// Mitsubishi GX Works2 project: shrimp_load_v02   PLC: FX3G
// Carga de PLC para monitoreo de piscina de camarones

PROGRAM MAIN
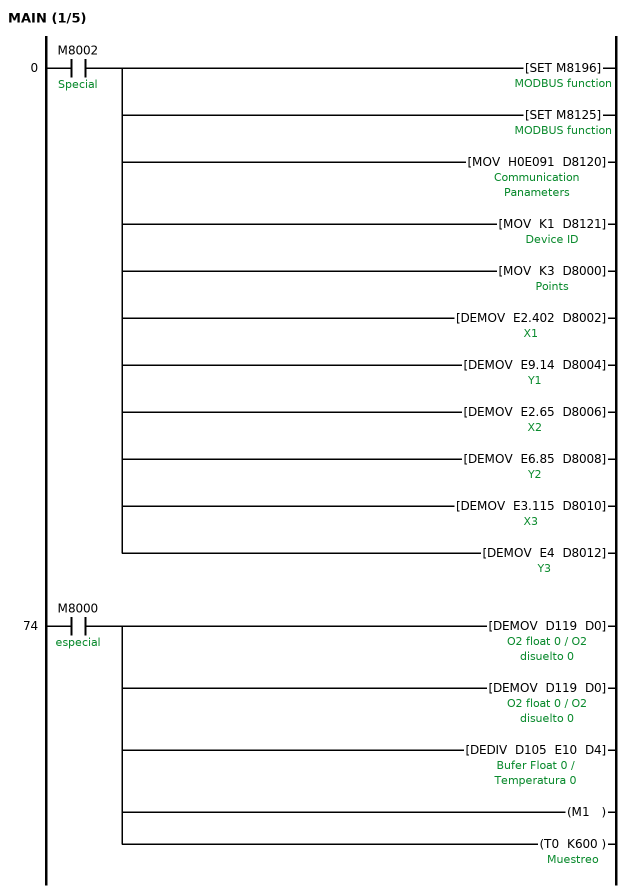
0     LD      M8002  ; Special
      SET     M8196  ; MODBUS function
      SET     M8125  ; MODBUS function
      MOV     H0E091 D8120  ; Communication Panameters
      MOV     K1 D8121  ; Device ID
      MOV     K3 D8000  ; Points
      DEMOV   E2.402 D8002  ; X1
      DEMOV   E9.14 D8004  ; Y1
      DEMOV   E2.65 D8006  ; X2
      DEMOV   E6.85 D8008  ; Y2
      DEMOV   E3.115 D8010  ; X3
      DEMOV   E4 D8012  ; Y3
74    LD      M8000  ; especial
      DEMOV   D119 D0  ; O2 float 0 / O2 disuelto 0
      DEMOV   D119 D0
      DEDIV   D105 E10 D4  ; Bufer Float 0 / Temperatura 0
      OUT     M1
      OUT     T0 K600  ; Muestreo
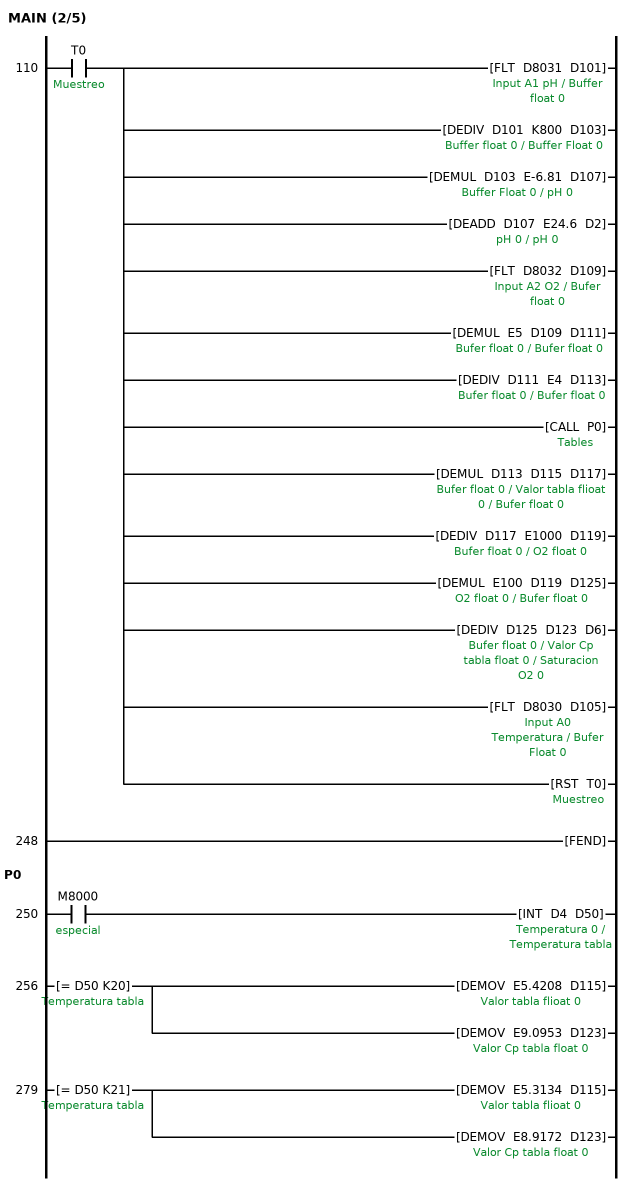
110   LD      T0  ; Muestreo
      FLT     D8031 D101  ; Input A1 pH / Buffer float 0
      DEDIV   D101 K800 D103  ; Buffer Float 0
      DEMUL   D103 E-6.81 D107  ; pH 0
      DEADD   D107 E24.6 D2  ; pH 0
      FLT     D8032 D109  ; Input A2 O2 / Bufer float 0
      DEMUL   E5 D109 D111  ; Bufer float 0
      DEDIV   D111 E4 D113  ; Bufer float 0
      CALL    P0  ; Tables
      DEMUL   D113 D115 D117  ; Valor tabla flioat 0 / Bufer float 0
      DEDIV   D117 E1000 D119
      DEMUL   E100 D119 D125  ; Bufer float 0
      DEDIV   D125 D123 D6  ; Valor Cp tabla float 0 / Saturacion O2 0
      FLT     D8030 D105  ; Input A0 Temperatura
      RST     T0  ; Muestreo
248   FEND
      P0
250   LD      M8000  ; especial
      INT     D4 D50  ; Temperatura tabla
256   LD=     D50 K20  ; Temperatura tabla
      DEMOV   E5.4208 D115
      DEMOV   E9.0953 D123
279   LD=     D50 K21  ; Temperatura tabla
      DEMOV   E5.3134 D115
      DEMOV   E8.9172 D123
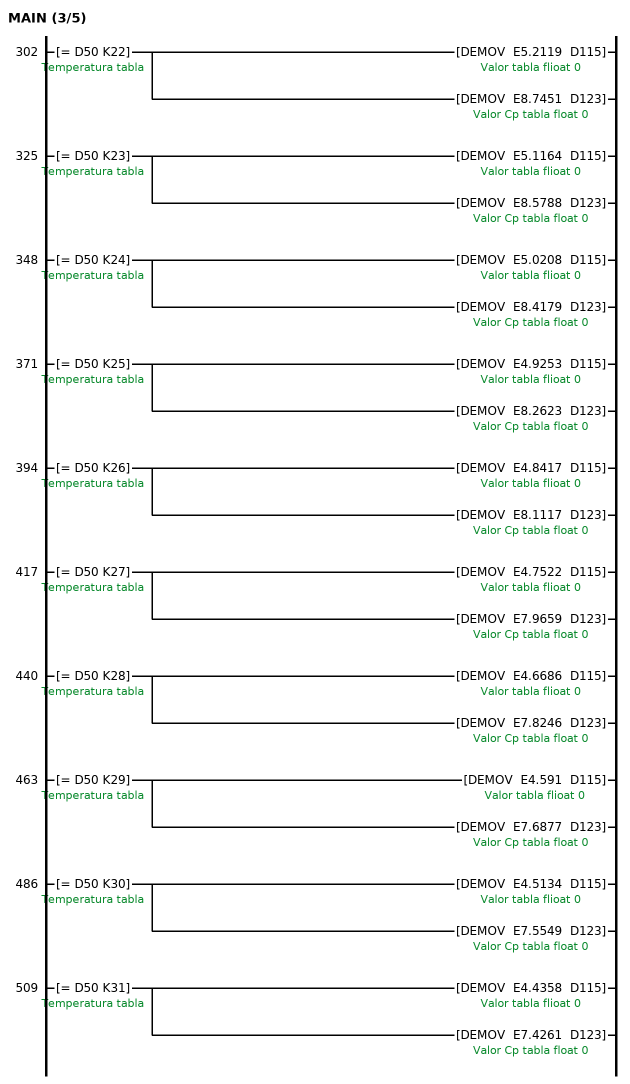
302   LD=     D50 K22  ; Temperatura tabla
      DEMOV   E5.2119 D115
      DEMOV   E8.7451 D123
325   LD=     D50 K23  ; Temperatura tabla
      DEMOV   E5.1164 D115
      DEMOV   E8.5788 D123
348   LD=     D50 K24  ; Temperatura tabla
      DEMOV   E5.0208 D115
      DEMOV   E8.4179 D123
371   LD=     D50 K25  ; Temperatura tabla
      DEMOV   E4.9253 D115
      DEMOV   E8.2623 D123
394   LD=     D50 K26  ; Temperatura tabla
      DEMOV   E4.8417 D115
      DEMOV   E8.1117 D123
417   LD=     D50 K27  ; Temperatura tabla
      DEMOV   E4.7522 D115
      DEMOV   E7.9659 D123
440   LD=     D50 K28  ; Temperatura tabla
      DEMOV   E4.6686 D115
      DEMOV   E7.8246 D123
463   LD=     D50 K29  ; Temperatura tabla
      DEMOV   E4.591 D115
      DEMOV   E7.6877 D123
486   LD=     D50 K30  ; Temperatura tabla
      DEMOV   E4.5134 D115
      DEMOV   E7.5549 D123
509   LD=     D50 K31  ; Temperatura tabla
      DEMOV   E4.4358 D115
      DEMOV   E7.4261 D123
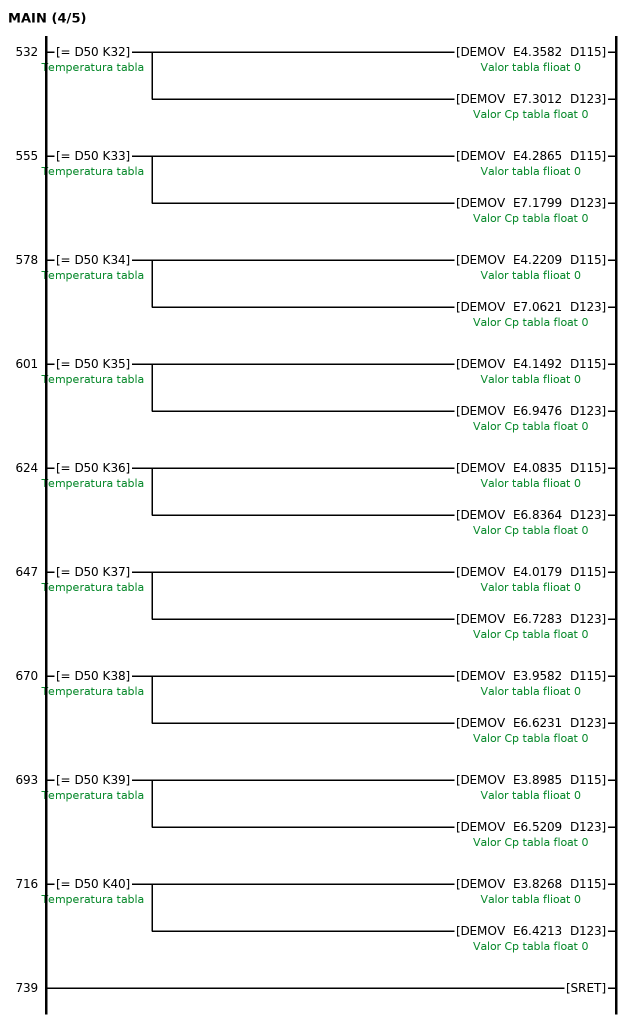
532   LD=     D50 K32  ; Temperatura tabla
      DEMOV   E4.3582 D115
      DEMOV   E7.3012 D123
555   LD=     D50 K33  ; Temperatura tabla
      DEMOV   E4.2865 D115
      DEMOV   E7.1799 D123
578   LD=     D50 K34  ; Temperatura tabla
      DEMOV   E4.2209 D115
      DEMOV   E7.0621 D123
601   LD=     D50 K35  ; Temperatura tabla
      DEMOV   E4.1492 D115
      DEMOV   E6.9476 D123
624   LD=     D50 K36  ; Temperatura tabla
      DEMOV   E4.0835 D115
      DEMOV   E6.8364 D123
647   LD=     D50 K37  ; Temperatura tabla
      DEMOV   E4.0179 D115
      DEMOV   E6.7283 D123
670   LD=     D50 K38  ; Temperatura tabla
      DEMOV   E3.9582 D115
      DEMOV   E6.6231 D123
693   LD=     D50 K39  ; Temperatura tabla
      DEMOV   E3.8985 D115
      DEMOV   E6.5209 D123
716   LD=     D50 K40  ; Temperatura tabla
      DEMOV   E3.8268 D115
      DEMOV   E6.4213 D123
739   SRET
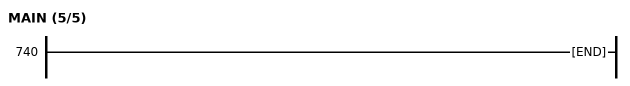
740   END
END_PROGRAM

// device comments not shown above
D1  ; O2 disuelto 1
D3  ; pH 1
D5  ; Temperatura 1
D7  ; Saturacion O2 1
D100  ; Buffer
D102  ; Buffer Float 1
D104  ; Bufer Float 1
D108  ; pH 1
D110  ; Bufer FLoat 1
D121  ; Bufer float 0
D127  ; Bufer float saturacion
D200  ; Buffer Float
D204  ; Bufer float
T200  ; Muestra
